(*
    This is the main program for execution of the unit tests.
    The program executes the test suites one after the other, with a delay of T#5S between
    each other (that is, as soon as one test suite has finished executing, the next
    one starts to execute immediately after). This delay is defined in the call to
    RUN_IN_SEQUENCE(T#5S).
    Within each test suite, the program executes each test one after the other, which
    is achieved by calling the TEST_ORDERED() for every test. The test-order is defined
    by the order of which the tests are being called.
    The tests include tests for function blocks which need several cycles to complete.
*)
PROGRAM PRG_TEST
VAR
    fbStateMachineFunctionBlock_Test : FB_StateMachineFunctionBlock_Test;
    fbTimedFunctionBlock_Test : FB_TimedFunctionBlock_Test;
END_VAR

TcUnit.RUN_IN_SEQUENCE(T#5S);

END_PROGRAM

(* stored: Version 1.1.0.1, ProductVersion 3.1.4022.18
   POU PRG_TEST: Id {01cac848-6a67-430a-a0cb-4e6885cf271a}, SpecialFunc None *)
